TYPE WinterShutdownParameters :
STRUCT
	EN: BOOL; // $(W1,S,R0)
	OutdoorTemperatureLimit: LREAL; // $(W1,S,R0)
END_STRUCT
END_TYPE

(* stored: Version 1.1.0.1, ProductVersion 3.1.4024.6
   DUT WinterShutdownParameters: Id {83b3717d-e33f-4162-9dbe-e6b865535ae6} *)
